FUNCTION _ARRAY_ABS : BOOL
VAR_INPUT
	pt : POINTER TO ARRAY[0..32000] OF REAL;
	size : UINT;
END_VAR
VAR
	i: UINT;
	stop: UINT;
END_VAR

(*
version 1.0	2. apr. 2008
programmer 	hugo
tested by	tobias

this function will calculate the absolute value of each element of the array and stroe the result instead of the element.
Array[i] := ABS(ARRAY[i]).
the function needs to be called:	array_avg(adr("array"),sizeof("array"));
because this function works with pointers its very time efficient and it needs no extra memory.

*)

stop := SHR(size,2)-1;
FOR i := 0 TO stop DO
	PT^[i] := ABS(PT^[i]);
END_FOR;
_ARRAY_ABS := TRUE;


(* revision history
hm	2. apr 2008		rev 1.0
	original version

*)

END_FUNCTION

(* stored: Version 1.1.0.1, ProductVersion 3.1.4022.7
   POU _ARRAY_ABS: Id {84ffc753-9bfd-40e9-b8aa-8fbd032815cd}, SpecialFunc None *)
